# EPICS alarm handler configuration: apps/alhConfig/beam_pos.alhConfig
GROUP    NULL                         BEAM_POSITION
CHANNEL  BEAM_POSITION                hallb_IPM2C21A_XPOS
$COMMAND  medm -x -attach -cmap -macro "sig=hallb_IPM2C21A_XPOS" aiaocalc_alarm.adl >> /dev/null
$ALARMCOUNTFILTER  10 120
$GUIDANCE
              The X beam position at nA BPM 2C21A is out of spec.  Inform MCC about this.
$END
CHANNEL  BEAM_POSITION                hallb_IPM2C21A_YPOS
$COMMAND  medm -x -attach -cmap -macro "sig=hallb_IPM2C21A_YPOS" aiaocalc_alarm.adl >> /dev/null
$ALARMCOUNTFILTER  10 120
$GUIDANCE
              The Y beam position at nA BPM 2C21A is out of spec.  Inform MCC about this.
$END
CHANNEL  BEAM_POSITION                hallb_IPM2C24A_XPOS
$COMMAND  medm -x -attach -cmap -macro "sig=hallb_IPM2C24A_XPOS" aiaocalc_alarm.adl >> /dev/null
$ALARMCOUNTFILTER  10 120
$GUIDANCE
              The X beam position at nA BPM 2C24A is out of spec.  Inform MCC about this.
$END
CHANNEL  BEAM_POSITION                hallb_IPM2C24A_YPOS
$COMMAND  medm -x -attach -cmap -macro "sig=hallb_IPM2C24A_YPOS" aiaocalc_alarm.adl >> /dev/null
$ALARMCOUNTFILTER  10 120
$GUIDANCE
              The Y beam position at nA BPM 2C24A is out of spec.  Inform MCC about this.
$END
CHANNEL  BEAM_POSITION                hallb_IPM2H00_XPOS
$COMMAND  medm -x -attach -cmap -macro "sig=hallb_IPM2H00_XPOS" aiaocalc_alarm.adl >> /dev/null
$ALARMCOUNTFILTER  10 120
$GUIDANCE
              The X beam position at nA BPM 2H00 is out of spec.  Inform MCC about this. Page Beamline expert if problem persists.
$END
CHANNEL  BEAM_POSITION                hallb_IPM2H00_YPOS
$COMMAND  medm -x -attach -cmap -macro "sig=hallb_IPM2H00_YPOS" aiaocalc_alarm.adl >> /dev/null
$ALARMCOUNTFILTER  10 120
$GUIDANCE
              The Y beam position at nA BPM 2H00 is out of spec.  Inform MCC about this. Page Beamline expert if problem persists.
$END
CHANNEL  BEAM_POSITION                hallb_IPM2H02_XPOS
$COMMAND  medm -x -attach -cmap -macro "sig=hallb_IPM2H02_XPOS" aiaocalc_alarm.adl >> /dev/null
$ALARMCOUNTFILTER  10 120
$GUIDANCE
              The X beam position at nA BPM 2H02 is out of spec.  Inform MCC about this. Page Beamline expert if problem persists.
$END
CHANNEL  BEAM_POSITION                hallb_IPM2H02_YPOS
$COMMAND  medm -x -attach -cmap -macro "sig=hallb_IPM2H02_YPOS" aiaocalc_alarm.adl >> /dev/null
$ALARMCOUNTFILTER  10 120
$GUIDANCE
              The Y beam position at nA BPM 2H02 is out of spec.  Inform MCC about this. Page Beamline expert if problem persists.
$END
